PROGRAM DoorLock
VAR
END_VAR

END_PROGRAM

(* stored: Version 1.1.0.1, ProductVersion 3.1.4024.11
   POU DoorLock: Id {9310e70f-f938-4312-bff5-999802aba96f}, SpecialFunc None *)
